{attribute 'qualified_only'}
{attribute 'to_string'}
TYPE E_LogType :
(
	invalid := 0,
	sysLog,
	auditLog,
	refuellingLog
) UDINT;
END_TYPE

(* stored: Version 1.1.0.1
   DUT E_LogType: Id {2b3efb61-c8a2-4327-b1c5-67f9013caacb} *)
